{attribute addProperty BoxType "EL3062-0000-0019"}
{attribute addProperty Id "AI_Standard_ChannelAT %I*ARRAY[0..1] OF AI_Standard_Channel_F16A160D6480WcStateAT %I*WcState_F855686C1620InfoDataAT %I*InfoData_BC63D37F80100"}
{attribute addProperty CRC "229822000"}
{attribute addProperty SizeInBites "160"}
{attribute addProperty SizeInBytes "20"}
TYPE EL3062_73C2997D :
STRUCT
	{attribute addProperty Name "AI_Standard_Channel"}
	AI_Standard_Channel : ARRAY[0..1] OF AI_Standard_Channel_F16A160D;
	{attribute addProperty Name "WcState"}
	WcState : WcState_F855686C;
	{attribute addProperty Name "InfoData"}
	InfoData : InfoData_BC63D37F;
END_STRUCT
END_TYPE

(* stored: Version 1.2.0.0, ProductVersion 3.1.4024.9
   DUT EL3062_73C2997D: Id {4650d8c0-d60a-4446-aba8-4082b0365b71} *)
